FUNCTION Band : LREAL
VAR_INPUT
	Value: lreal;
	Target: LREAL;
	Width: LREAL;
END_VAR
VAR
END_VAR

  Band := LimitValue(Value - Target, -Width, Width) / Width;

END_FUNCTION

(* stored: Version 1.1.0.1, ProductVersion 3.1.4024.3
   POU Band: Id {ef86ebae-c3fa-4ff1-aa85-67b542bf726e}, SpecialFunc None *)
